TYPE ST_EM_HMI :
	STRUCT
		Cmd : ST_EM_Cmd;
		Cfg : ST_EM_Cfg;
		Sts : ST_EM_Sts;
	END_STRUCT
END_TYPE

(* stored: Version 1.1.0.1, ProductVersion 3.1.4024.12
   DUT ST_EM_HMI: Id {b0a650bc-7971-419d-9284-c263ab10de8f} *)
